(* PLC project management, Dassault Systèmes ControlBuild 2024x Refresh1 *)
(* stored: creationDateTime 2024-04-12T14:05:57-01:00 *)

FUNCTION_BLOCK copie_batch.management
  VAR_INPUT
    cycleInProgress : BOOL := false;
    endCycleRequest : BOOL := false;
    kneadingOk : BOOL := false;
    syrupWeighingOk : BOOL := false;
    flourWeighingOk : BOOL := false;
  END_VAR
  VAR_OUTPUT
    cycleEnd : BOOL := false;
    flourWeighingRq : BOOL := false;
    syrupWeighingRq : BOOL := false;
    kneadingRq : BOOL := false;
  END_VAR

INITIAL_STEP 10:
  COMPUTE_FUNCTION_BLOCKS(S);
END_STEP
TRANSITION FROM 10 TO 11
  := cycleInProgress;
END_TRANSITION
STEP 11:
  11_INLINE1(N);
END_STEP
ACTION 11_INLINE1:
  flourWeighingRq;
END_ACTION
TRANSITION FROM 11 TO 12
  := flourWeighingOk AND cycleInProgress;
END_TRANSITION
STEP 12:
  12_INLINE2(N);
END_STEP
ACTION 12_INLINE2:
  kneadingRq;
  syrupWeighingRq;
END_ACTION
TRANSITION FROM 12 TO 13
  := syrupWeighingOk AND cycleInProgress;
END_TRANSITION
STEP 13:
END_STEP
TRANSITION FROM 13 TO 14
  := kneadingOk AND cycleInProgress;
END_TRANSITION
STEP 14:
  14_INLINE3(N);
END_STEP
ACTION 14_INLINE3:
  IF endCycleRequest THEN
  	cycleEnd;
  END_IF;
END_ACTION
TRANSITION FROM 14 TO 10
  := TRUE;
END_TRANSITION
ACTION COMPUTE_FUNCTION_BLOCKS:  (* blocks drawn on the SFC sheet *)
  G1:
END_ACTION
END_FUNCTION_BLOCK
